{attribute 'qualified_only'}
VAR_GLOBAL
END_VAR

(* stored: Version 1.1.0.1, ProductVersion 3.1.4022.7
   GVL GVL_05_Manual_Servo_Motor_Shelf_Z: Id {d6edbbb1-f422-4e2e-b384-60bfc0ee9507} *)
